TYPE EtcMasterBase_62654B43 : 
STRUCT
END_STRUCT
END_TYPE

(* stored: Version 1.1.0.1, ProductVersion 3.1.4024.9
   DUT EtcMasterBase_62654B43: Id {07b646bf-3927-04c3-3917-586daf277db7} *)
